// TwinCAT 3 PLC project tank1
// ProgramVersion: 3.1.4023.0
// libraries:
//   Tc2_Standard, * (Beckhoff Automation GmbH)
//   Tc2_System, * (Beckhoff Automation GmbH)
//   Tc3_Module, * (Beckhoff Automation GmbH)
// project tree:
//   / PlcTask.TcTTO
//   POUs/ MAIN.TcPOU, Tank1.TcPOU, Tank1_1.TcPOU, Tank1_1_1.TcPOU
// real-time tasks:
//   TASK PlcTask: cycle T#10ms, priority 20, ADS port 350

CONFIGURATION tank1
    RESOURCE PLC ON TwinCAT3
        TASK PlcTask(INTERVAL := T#10ms, PRIORITY := 20);
        PROGRAM MAIN WITH PlcTask : MAIN;
    END_RESOURCE
END_CONFIGURATION

// ---- POUs/MAIN.TcPOU
PROGRAM MAIN
VAR
	//tank : tank1;
	//tank : Tank1_1;
	tank : Tank1_1_1;
	bfill : BOOL;
 
END_VAR


tank(bSwitchFill := bfill);

END_PROGRAM

// ---- POUs/Tank1_1_1.TcPOU
FUNCTION_BLOCK Tank1_1_1
VAR_INPUT
	//bSwitchFill : BOOL;
	bSwitchSink : BOOL;
END_VAR
VAR_IN_OUT
	bSwitchFill : BOOL;
END_VAR
VAR_OUTPUT
END_VAR
VAR
	bShl : BOOL := FALSE;
	bSll : BOOL := TRUE;
	bS90l : BOOL;
	nState : INT;
	level: INT := 3;
	tTime : TON;
	rTrig : R_TRIG;	
	
END_VAR


IF level < 5 THEN
	bShl := FALSE;	
	bS90l := TRUE;
	bSll := TRUE;
ELSIF level >= 5 AND level < 90 THEN
	bShl := FALSE;	
	bS90l := TRUE;
	bSll := FALSE;
ELSIF level >= 90 AND level < 100 THEN
	bShl := FALSE;	
	bS90l := FALSE;
	bSll := FALSE;
ELSIF level = 100 THEN
	bShl := TRUE;	
	bS90l := FALSE;
	bSll := FALSE;
END_IF




CASE nState OF
	
	0:	
		IF  NOT bSwitchSink THEN
			IF bSll THEN
				bSwitchFill := TRUE;
			END_IF
			tTime(IN := bSwitchFill,PT := T#2S);
			rTrig(CLK := tTime.Q);
			IF rTrig.Q THEN
				level := level + 2;
				tTime(IN := FALSE);
				IF bShl THEN
					bSwitchFill := FALSE;
					nState := 10;
				END_IF
			END_IF
		 		
		ELSE
			IF NOT bSwitchFill THEN
				nState := 10;
			ELSE
				IF bSll THEN
					bSwitchFill := TRUE;
				END_IF
				tTime(IN := bSwitchFill,PT := T#2S);
				rTrig(CLK := tTime.Q);
				IF rTrig.Q THEN
					level := level + 1;
					tTime(IN := FALSE);
					IF bShl THEN
						bSwitchFill := FALSE;
						nState := 10;
					END_IF
				END_IF
			END_IF
		END_IF
		
	10: 
		IF  bSwitchSink THEN
			IF bShl OR NOT bS90l THEN
				bSwitchFill := FALSE;
			ELSE
				bSwitchFill := bSwitchFill;
			END_IF
			IF NOT bSwitchFill THEN
				tTime(IN := bSwitchSink,PT := T#2S);
				rTrig(CLK := tTime.Q);
				IF rTrig.q THEN
					tTime(IN := FALSE);
					level := level - 1;
					IF bSll THEN
						bSwitchSink := FALSE;
						nState := 0;
					END_IF
				END_IF
			ELSE
				nState := 0;
			END_IF
		ELSE
			IF NOT bSwitchFill THEN
				nState := 10;
			ELSE
				nState := 0;
			END_IF		
		END_IF
					
END_CASE

END_FUNCTION_BLOCK

// ---- POUs/Tank1.TcPOU
FUNCTION_BLOCK Tank1
VAR_INPUT
	//bSwitchFill : BOOL;
	bSwitchSink : BOOL;
END_VAR
VAR_IN_OUT
	bSwitchFill : BOOL;
END_VAR
VAR_OUTPUT
END_VAR
VAR
	bShl : BOOL := FALSE;
	bSll : BOOL := TRUE;
	nState : INT;
	level: INT := 5;
	tTime1 : TON;
	tTime2 : TON;
	rTrig1 : R_TRIG;
	rTrig2 : R_TRIG;
	
	
END_VAR


CASE nState OF
	0:	
		
		IF  NOT bSwitchSink THEN
			IF bSll THEN
				bSwitchFill := TRUE;
			END_IF
			tTime1(IN := bSwitchFill,PT := T#2S);
			rTrig1(CLK := tTime1.Q);
			IF rTrig1.Q THEN
				level := level + 1;
				tTime1(IN := FALSE);
				IF level = 100 THEN
				bShl := TRUE;
				bSll := FALSE;	
				bSwitchFill := FALSE;
				nState := 10;
				END_IF
			END_IF
		
 		
		ELSIF  bSwitchSink THEN
			IF bSll THEN
				bSwitchFill := TRUE;
			END_IF
			tTime1(IN := bSwitchFill,PT := T#3S);
			rTrig1(CLK := tTime1.Q);
			IF rTrig1.Q THEN
				level := level + 1;
				tTime1(IN := FALSE);
				IF level = 100 THEN
				bShl := TRUE;
				bSll := FALSE;
				bSwitchFill := FALSE;
				nState := 10;
				END_IF
			END_IF
		END_IF
		
	10: 
		
		IF  bSwitchSink  THEN
			IF bShl AND level > 90 THEN
				bSwitchFill := FALSE;
				tTime2(IN := bSwitchSink,PT := T#1S);
				rTrig2(CLK := tTime2.Q);
				IF rTrig2.q THEN
				tTime2(IN := FALSE);
				level := level - 1;
				IF level = 5 THEN
				bSwitchSink := FALSE;
				bShl := FALSE;
				bSll := TRUE;
				nState := 0;
				END_IF
				END_IF
			ELSIF level <= 90 THEN
					IF bSwitchFill THEN
					
						tTime2(IN := bSwitchSink,PT := T#3S);
						rTrig2(CLK := tTime2.Q);
						IF rTrig2.q THEN
						tTime2(IN := FALSE);
						level := level + 1;
						IF level = 100 THEN
						bSwitchSink := FALSE;
						bShl := TRUE;
						bSll := FALSE;
						nState := 10;
						END_IF
						END_IF
						
					ELSE
						tTime2(IN := bSwitchSink,PT := T#1S);
						rTrig2(CLK := tTime2.Q);
						IF rTrig2.q THEN
						tTime2(IN := FALSE);
						level := level - 1;
						IF level = 5 THEN
						bSwitchSink := FALSE;
						bShl := FALSE;
						bSll := TRUE;
						nState := 0;
						END_IF
						END_IF
						
					END_IF
			
			END_IF		
			
			
		END_IF
		
		
END_CASE

END_FUNCTION_BLOCK

// ---- POUs/Tank1_1.TcPOU
FUNCTION_BLOCK Tank1_1
VAR_INPUT
	//bSwitchFill : BOOL;
	bSwitchSink : BOOL;
END_VAR
VAR_IN_OUT
	bSwitchFill : BOOL;
END_VAR
VAR_OUTPUT
END_VAR
VAR
	bShl : BOOL := FALSE;
	bSll : BOOL := TRUE;
	nState : INT;
	level: INT := 3;
	tTime : TON;
	rTrig : R_TRIG;	
	
END_VAR



CASE nState OF
	
	0:	
		IF  NOT bSwitchSink THEN
			IF bSll THEN
				bSwitchFill := TRUE;
			END_IF
			(*IF NOT bShl THEN
				bSwitchFill := TRUE;
			END_IF*)
			tTime(IN := bSwitchFill,PT := T#1S);
			rTrig(CLK := tTime.Q);
			IF rTrig.Q THEN
				level := level + 2;
				tTime(IN := FALSE);
				IF level >= 5 THEN
					bSll := FALSE;
				END_IF
				IF level = 100 THEN
					bShl := TRUE;
					bSwitchFill := FALSE;
					nState := 10;
				END_IF
			END_IF
		 		
		ELSE
			IF NOT bSwitchFill THEN
				nState := 10;
			ELSE
				IF bSll THEN
					bSwitchFill := TRUE;
				END_IF
				(*IF NOT bShl THEN
					bSwitchFill := TRUE;
				END_IF*)
				tTime(IN := bSwitchFill,PT := T#1S);
				rTrig(CLK := tTime.Q);
				IF rTrig.Q THEN
					level := level + 1;
					tTime(IN := FALSE);
					IF level >= 5 THEN
						bSll := FALSE;
					END_IF
					IF level = 100 THEN
						bShl := TRUE;
						bSwitchFill := FALSE;
						nState := 10;
					END_IF
				END_IF
			END_IF
		END_IF
		
	10: 
		
		IF  bSwitchSink THEN
			IF bShl THEN
				bSwitchFill := FALSE;
			END_IF
			IF level > 90 THEN
				bSwitchFill := FALSE;
			ELSIF level <= 90 THEN
				bSwitchFill := bSwitchFill;
			END_IF
			IF NOT bSwitchFill THEN
				tTime(IN := bSwitchSink,PT := T#1S);
				rTrig(CLK := tTime.Q);
				IF rTrig.q THEN
					tTime(IN := FALSE);
					level := level - 1;
					IF level <> 100 THEN
						bShl := FALSE;
					END_IF
					IF level < 5 THEN
						bSwitchSink := FALSE;
						bSll := TRUE;
						nState := 0;
					END_IF
				END_IF
			ELSE
				IF level <> 100 THEN
					bShl := FALSE;
				END_IF
				nState := 0;
			END_IF
		ELSE
			IF NOT bSwitchFill THEN
				nState := 10;
			ELSE
				nState := 0;
			END_IF		
		END_IF
					
END_CASE

END_FUNCTION_BLOCK
